(* PLC project 未命名, 未知 未命名 1 *)
(* stored: creationDateTime 2020-04-08T00:09:48, modificationDateTime 2020-10-02T14:55:35 *)

PROGRAM program0
  VAR
    DelayTime : TIME := T#5s;  (* 每轮时间，T#5s=延时5秒 *)
    Bad : BOOL := false;  (* 异常 *)
    Good : BOOL := true;  (* 正常 *)
    Closed : BOOL := true;  (* 是否要关闭，T=是|F=否 *)
    Open : BOOL := false;  (* 是否要打开，T=是|F=否 *)
    CriticalFMValue : REAL := 0.5;  (* 频率差值 *)
    CriticalRange : REAL := 49.9;  (* 频率阈值 *)
    CriticalTemp : REAL := 50.0;  (* 温度阈值 *)
    CriticalLoadingValue : REAL := 100.0;  (* 负载阈值 *)
    fm : REAL := 50.0;
    TON0 : TON;
    WaitStatus : BOOL := true;
    pass_code : BOOL;
  END_VAR
  VAR
    line_cb_0 AT %QX00.0 : BOOL;
    line_cb_1 AT %QX00.1 : BOOL;
    line_cb_2 AT %QX00.2 : BOOL;
    line_cb_3 AT %QX00.3 : BOOL;
    line_cb_4 AT %QX00.4 : BOOL;
    line_cb_5 AT %QX00.5 : BOOL;
    line_cb_6 AT %QX00.6 : BOOL;
    line_cb_7 AT %QX00.7 : BOOL;
    line_cb_8 AT %QX00.8 : BOOL;
    line_cb_9 AT %QX00.9 : BOOL;
    line_cb_10 AT %QX00.10 : BOOL;
    line_cb_11 AT %QX00.11 : BOOL;
    line_cb_12 AT %QX00.12 : BOOL;
    line_cb_13 AT %QX00.13 : BOOL;
    line_cb_14 AT %QX00.14 : BOOL;
    line_cb_15 AT %QX00.15 : BOOL;
    line_cb_16 AT %QX00.16 : BOOL;
    line_cb_17 AT %QX00.17 : BOOL;
    relay_0 AT %QX00.100 : BOOL;
    relay_1 AT %QX00.101 : BOOL;
    relay_2 AT %QX00.102 : BOOL;
    relay_3 AT %QX00.103 : BOOL;
    line_loading_0 AT %MD0 : REAL;
    line_loading_1 AT %MD1 : REAL;
    line_loading_2 AT %MD2 : REAL;
    line_loading_3 AT %MD3 : REAL;
    line_loading_4 AT %MD4 : REAL;
    line_loading_5 AT %MD5 : REAL;
    line_loading_6 AT %MD6 : REAL;
    line_loading_7 AT %MD7 : REAL;
    line_loading_8 AT %MD8 : REAL;
    line_loading_9 AT %MD9 : REAL;
    line_loading_10 AT %MD10 : REAL;
    line_loading_11 AT %MD11 : REAL;
    line_loading_12 AT %MD12 : REAL;
    line_loading_13 AT %MD13 : REAL;
    line_loading_14 AT %MD14 : REAL;
    line_loading_15 AT %MD15 : REAL;
    line_loading_16 AT %MD16 : REAL;
    line_loading_17 AT %MD17 : REAL;
    line_load_percent_0 AT %MD400 : REAL;
    line_load_percent_1 AT %MD401 : REAL;
    line_load_percent_2 AT %MD402 : REAL;
    line_load_percent_3 AT %MD403 : REAL;
    line_load_percent_4 AT %MD404 : REAL;
    line_load_percent_5 AT %MD405 : REAL;
    line_load_percent_6 AT %MD406 : REAL;
    line_load_percent_7 AT %MD407 : REAL;
    line_load_percent_8 AT %MD408 : REAL;
    line_load_percent_9 AT %MD409 : REAL;
    line_load_percent_10 AT %MD410 : REAL;
    line_load_percent_11 AT %MD411 : REAL;
    line_load_percent_12 AT %MD412 : REAL;
    line_load_percent_13 AT %MD413 : REAL;
    line_load_percent_14 AT %MD414 : REAL;
    line_load_percent_15 AT %MD415 : REAL;
    line_load_percent_16 AT %MD416 : REAL;
    line_load_percent_17 AT %MD417 : REAL;
    loads_0 AT %MD100 : REAL;
    loads_1 AT %MD101 : REAL;
    loads_2 AT %MD102 : REAL;
    loads_3 AT %MD103 : REAL;
    loads_4 AT %MD104 : REAL;
    loads_5 AT %MD105 : REAL;
    loads_6 AT %MD106 : REAL;
    loads_7 AT %MD107 : REAL;
    loads_8 AT %MD108 : REAL;
    loads_9 AT %MD109 : REAL;
    transformer_temp_0 AT %QX00.50 : BOOL;
    transformer_temp_1 AT %QX00.51 : BOOL;
    fm_0 AT %MD300 : REAL;
    fm_1 AT %MD301 : REAL;
    fm_2 AT %MD302 : REAL;
    fm_3 AT %MD303 : REAL;
    fm_show AT %MD304 : REAL;
  END_VAR

            (* Auto-transfer *)
IF line_cb_0 = Open THEN
  IF relay_0 = Good THEN
  line_cb_16 := Closed;
  END_IF;
END_IF;

IF line_cb_1 = Open THEN
  IF relay_1 = Good THEN
    line_cb_16 := Closed;
  END_IF;
END_IF;



(*Transformer Overheating Protection *)
IF transformer_temp_0 = Bad THEN
  line_cb_4 := Open;
  line_cb_5 := Open;
END_IF;

IF transformer_temp_1 = Bad THEN
  line_cb_12 := Open;
  line_cb_13 := Open;
END_IF;

IF line_cb_5 = Open THEN
  line_cb_4 := Open;
END_IF;

IF line_cb_13 = Open THEN
  line_cb_12 := Open;
END_IF;

(*Relay Isolation*
IF relay_2 = Bad THEN
  line_cb_5 := Open;
  line_cb_17 := Open;
END_IF;

IF relay_3 = Bad THEN
  line_cb_13 := Open;
  line_cb_17 := Open;
END_IF;
*)



(*Overcurrent Protection*)
IF line_load_percent_0 >= CriticalLoadingValue THEN
    line_cb_0 := Open;
END_IF;

IF line_load_percent_1 >= CriticalLoadingValue THEN
    line_cb_1 := Open;
END_IF;

IF line_load_percent_2 >= CriticalLoadingValue THEN
    line_cb_2 := Open;
END_IF;

IF line_load_percent_3 >= CriticalLoadingValue THEN
    line_cb_3 := Open;
END_IF;

IF line_load_percent_4 >= CriticalLoadingValue THEN
    line_cb_4 := Open;
END_IF;

IF line_load_percent_5 >= CriticalLoadingValue THEN
    line_cb_5 := Open;
END_IF;

IF line_load_percent_6 >= CriticalLoadingValue THEN
    line_cb_6 := Open;
END_IF;

IF line_load_percent_7 >= CriticalLoadingValue THEN
    line_cb_7 := Open;
END_IF;

IF line_load_percent_8 >= CriticalLoadingValue THEN
    line_cb_8 := Open;
END_IF;

IF line_load_percent_9 >= CriticalLoadingValue THEN
    line_cb_9 := Open;
END_IF;

IF line_load_percent_10 >= CriticalLoadingValue THEN
    line_cb_10 := Open;
END_IF;

IF line_load_percent_11 >= CriticalLoadingValue THEN
    line_cb_11 := Open;
END_IF;

IF line_load_percent_12 >= CriticalLoadingValue THEN
    line_cb_12 := Open;
END_IF;

IF line_load_percent_13 >= CriticalLoadingValue THEN
    line_cb_13 := Open;
END_IF;

IF line_load_percent_14 >= CriticalLoadingValue THEN
    line_cb_14 := Open;
END_IF;

IF line_load_percent_15 >= CriticalLoadingValue THEN
    line_cb_15 := Open;
END_IF;

IF line_load_percent_16 >= CriticalLoadingValue THEN
    line_cb_16 := Open;
END_IF;

IF line_load_percent_17 >= CriticalLoadingValue THEN
    line_cb_17 := Open;
END_IF;
          
END_PROGRAM

CONFIGURATION Config0
  RESOURCE Res0 ON PLC
    TASK task0(INTERVAL := T#20ms, PRIORITY := 0);
    PROGRAM instance0 WITH task0 : program0;
  END_RESOURCE
END_CONFIGURATION
